// TIA Portal V20 export
FUNCTION_BLOCK "AdjRight"   // FB530, FBD
{ S7_Optimized_Access := 'TRUE' }
// stored: AutoNumber false, MemoryReserve 100, SetENOAutomatically false
   VAR
      Var { ExternalAccessible := 'False'; ExternalVisible := 'False'; ExternalWritable := 'False'} : "TypeVar";
      Cmd { ExternalAccessible := 'False'; ExternalVisible := 'False'; ExternalWritable := 'False'} : "TypeCmd";
      Enc { ExternalAccessible := 'False'; ExternalVisible := 'False'; ExternalWritable := 'False'} : "SysCounterFast";
      Pos { ExternalAccessible := 'False'; ExternalVisible := 'False'; ExternalWritable := 'False'} : "SysPos";
      AdjSlow { ExternalAccessible := 'False'; ExternalVisible := 'False'; ExternalWritable := 'False'} : "SysMotor";
      AdjFast { ExternalAccessible := 'False'; ExternalVisible := 'False'; ExternalWritable := 'False'} : "SysLinMotC1150";
      TAutoOn { ExternalAccessible := 'False'; ExternalVisible := 'False'; ExternalWritable := 'False'} : TON_TIME;
      TAutoTarPosManOn { ExternalAccessible := 'False'; ExternalVisible := 'False'; ExternalWritable := 'False'} : TON_TIME;
      T { ExternalAccessible := 'False'; ExternalVisible := 'False'; ExternalWritable := 'False'} : Array[1..5] of IEC_TIMER;
      adjFastPnSlaveOff { ExternalAccessible := 'False'; ExternalVisible := 'False'; ExternalWritable := 'False'} : "SysPnSlaveDeactivate";
      tarOld { ExternalAccessible := 'False'; ExternalVisible := 'False'; ExternalWritable := 'False'} : DInt;
      autoTarPosMan { ExternalAccessible := 'False'; ExternalVisible := 'False'; ExternalWritable := 'False'} : Bool;
      setValueEnc { ExternalAccessible := 'False'; ExternalVisible := 'False'; ExternalWritable := 'False'} : Bool;
      autoRef { ExternalAccessible := 'False'; ExternalVisible := 'False'; ExternalWritable := 'False'} : Bool;
      posOld { ExternalAccessible := 'False'; ExternalVisible := 'False'; ExternalWritable := 'False'} : Real;
      posDiff { ExternalAccessible := 'False'; ExternalVisible := 'False'; ExternalWritable := 'False'} : Real;
   END_VAR
   VAR_TEMP
      CtrlPc : Struct
         ackErr : Bool;
         manModeActive : Bool;
         manP : Bool;
         manM : Bool;
         manRefRun : Bool;
      END_STRUCT;
      CtrlLinMot : Struct
         mode : Int;
         target : Real;
         speed : Real;
         acc : Real;
         dec : Real;
         jerk : Real;
         autoRef : Bool;
      END_STRUCT;
      refPosDiff : DInt;
      offsetNoStd : Real;
      refPosDiffCalib : DInt;
      modeCalib : Int;
      disMechanicToZero : Int;   // distance mechanic part right to zero [mm]
   END_VAR
   VAR_TEMP   // added for the SCL form of the ladder/FBD networks
      _w1 : Bool;
   END_VAR
BEGIN

REGION Network 1 (SCL): offset for no standard calibration
   (* 
   normally the distance from camera to board should be 550mm
   for special application the distance is different
   the distance can be changed in the goldeneye program
   if its different then 550mm a offset will be added
   *)
   #offsetNoStd := 0.0;
   IF "ComRd".Data.Right.RefPosToBoard <> 550 THEN
       #offsetNoStd := (DINT_TO_REAL("ComRd".Data.Right.RefPosToBoard) - 550.0);
   ELSE
       #offsetNoStd := 0.0;
   END_IF;
END_REGION

REGION Network 2 (SCL): calibration value for offset
   (* 
   modus for calibartion
   camera must be referenced first
   mode 1 -->   the camera must be moved manually to position 550mm from board and
                 then press "Set Nullpoint"
   mode 2 -->   the camera must be moved to a other position and
                 then must be measured from the calibration tool to the camera and
                 this value must be putted in after pressing "Set Nullpoint"
   *)         
   #disMechanicToZero := 870; 
   #modeCalib := 2;
   IF #modeCalib = 1 THEN
       #refPosDiffCalib := "ComRd".Data.Right.TargetPos;
   ELSIF #modeCalib = 2 THEN
       #refPosDiffCalib := (#disMechanicToZero * 10) - ("ComRd".Data.Right.CalibratePos + 5500);
   END_IF;
END_REGION

REGION Network 3 (SCL): calibration value from pc
   "ComSd".Data.Right.SetCalibratePosOk := FALSE;

   IF "ComRd".Data.Right.SetCalibratePos THEN

       IF "G".Cfg.adjRightActive THEN
           #refPosDiff := REAL_TO_DINT("Enc"."8BC1.R".act * 10.0) - #refPosDiffCalib;
       ELSIF "G".Cfg.adjRightActiveLinMot THEN
           #refPosDiff := REAL_TO_DINT("Enc"."8U1.R".act * 10.0) - #refPosDiffCalib;
       END_IF;

       "Ref".adjRightCalOffset := #refPosDiff;
       "ComSd".Data.Right.SetCalibratePosOk := TRUE;

   END_IF;
END_REGION

REGION Network 4 (SCL): target position
   #Cmd.target := "G".Batch.width / 2.0;
   IF "G".Cfg.modeBoardPassing = 1 AND ("G".Cfg.modeDimension = 2 OR "G".Cfg.modeDimension = 4) AND NOT "G".Batch.stdActive THEN
       #Cmd.target := "G".Batch.width / 2.0 + ("G".Batch.widthMeasure - "G".Batch.width);
   END_IF;

   IF "G".Cfg.modeBoardPassing = 3 AND ("G".Cfg.modeDimension = 2 OR "G".Cfg.modeDimension = 4) AND NOT "G".Batch.stdActive THEN
       #Cmd.target :=  "G".Batch.senRightVal;
   END_IF;

   IF #autoTarPosMan THEN
       #Cmd.target := DINT_TO_REAL("ComRd".Data.Right.TargetPos) / 10.0;
   END_IF;

   "Ref".adjRightTar := #Cmd.target + (DINT_TO_REAL("Ref".adjRightCalOffset) / 10.0) + #offsetNoStd - "Enc"."8B1.B".offset;
END_REGION

REGION Network 5 (SCL): data from pc
   IF NOT "G".errComPc THEN
       #CtrlPc.manModeActive := "ComRd".Data.Right.ManModeActive;
       #CtrlPc.manP := "ComRd".Data.Right.ManPlus;
       #CtrlPc.manM := "ComRd".Data.Right.ManMinus;
       #CtrlPc.manRefRun := "ComRd".Data.Right.ManRefRun;
   ELSE
       #CtrlPc.manModeActive := TRUE;
       #CtrlPc.manP := FALSE;
       #CtrlPc.manM := FALSE;
       #CtrlPc.manRefRun := FALSE;
   END_IF;
   #CtrlPc.ackErr := "G".ack;
END_REGION

REGION Network 6: off
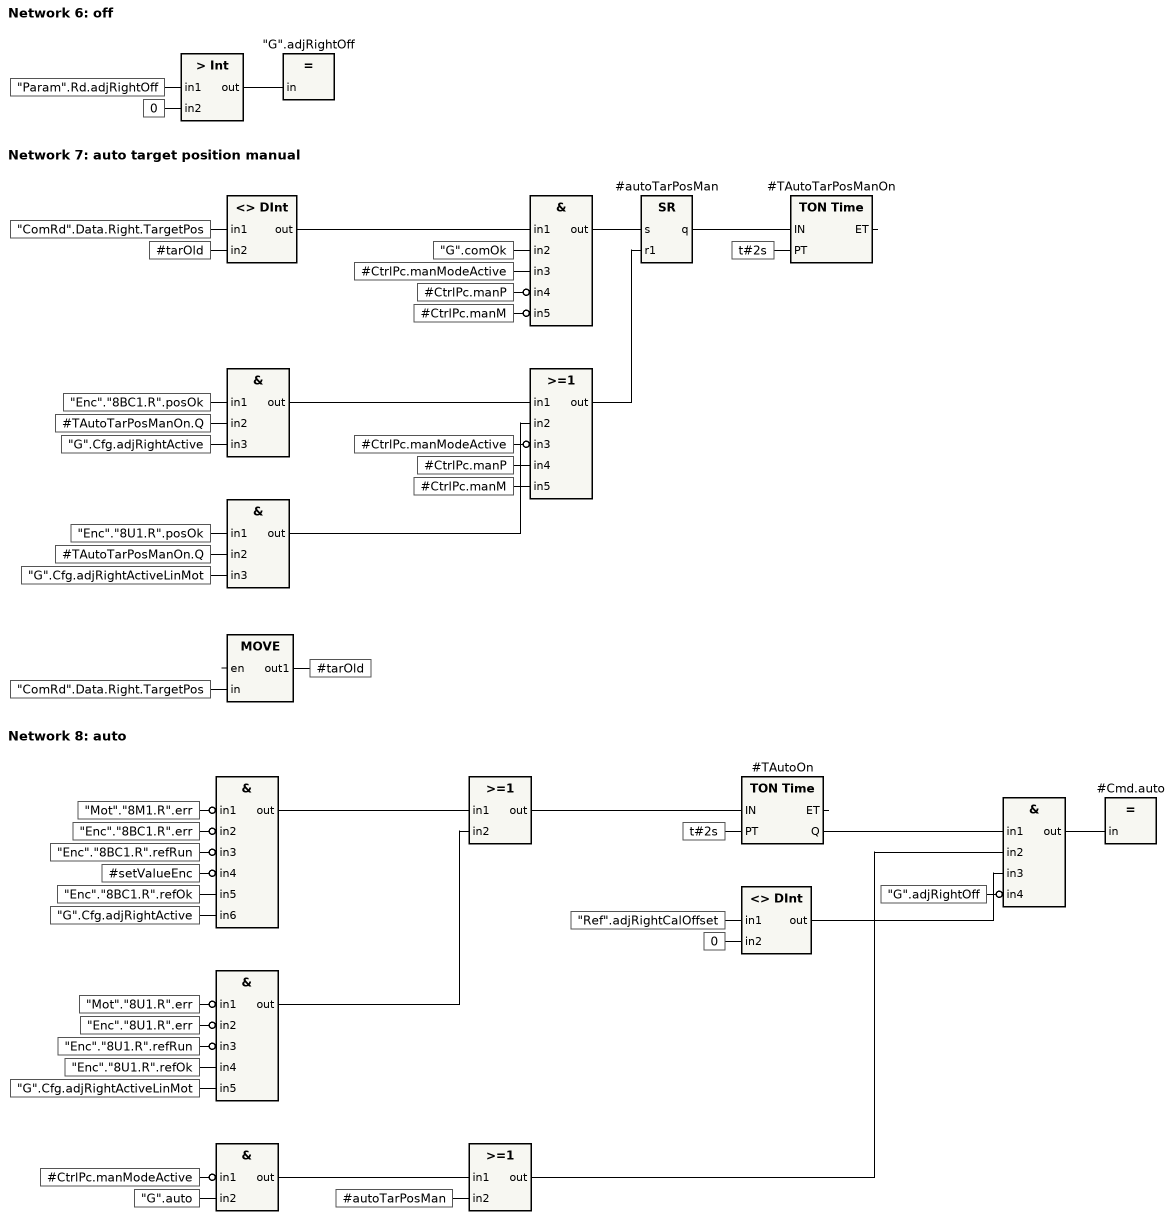
   "G".adjRightOff := "Param".Rd.adjRightOff > 0;
END_REGION

REGION Network 7: auto target position manual
   IF ("ComRd".Data.Right.TargetPos <> #tarOld) AND "G".comOk AND #CtrlPc.manModeActive AND NOT #CtrlPc.manP AND NOT #CtrlPc.manM THEN
       #autoTarPosMan := TRUE;   // SR flip-flop
   END_IF;
   IF ("Enc"."8BC1.R".posOk AND #TAutoTarPosManOn.Q AND "G".Cfg.adjRightActive) OR ("Enc"."8U1.R".posOk AND #TAutoTarPosManOn.Q AND "G".Cfg.adjRightActiveLinMot) OR NOT #CtrlPc.manModeActive OR #CtrlPc.manP OR #CtrlPc.manM THEN
       #autoTarPosMan := FALSE;
   END_IF;
   #TAutoTarPosManOn(IN := #autoTarPosMan, PT := t#2s);   // TON
   #tarOld := "ComRd".Data.Right.TargetPos;
END_REGION

REGION Network 8: auto
   #TAutoOn(IN := (NOT "Mot"."8M1.R".err AND NOT "Enc"."8BC1.R".err AND NOT "Enc"."8BC1.R".refRun AND NOT #setValueEnc AND "Enc"."8BC1.R".refOk AND "G".Cfg.adjRightActive) OR (NOT "Mot"."8U1.R".err AND NOT "Enc"."8U1.R".err AND NOT "Enc"."8U1.R".refRun AND "Enc"."8U1.R".refOk AND "G".Cfg.adjRightActiveLinMot),   // TON
            PT := t#2s);
   #Cmd.auto := #TAutoOn.Q AND ((NOT #CtrlPc.manModeActive AND "G".auto) OR #autoTarPosMan) AND ("Ref".adjRightCalOffset <> 0) AND NOT "G".adjRightOff;
END_REGION

REGION Network 9: manual
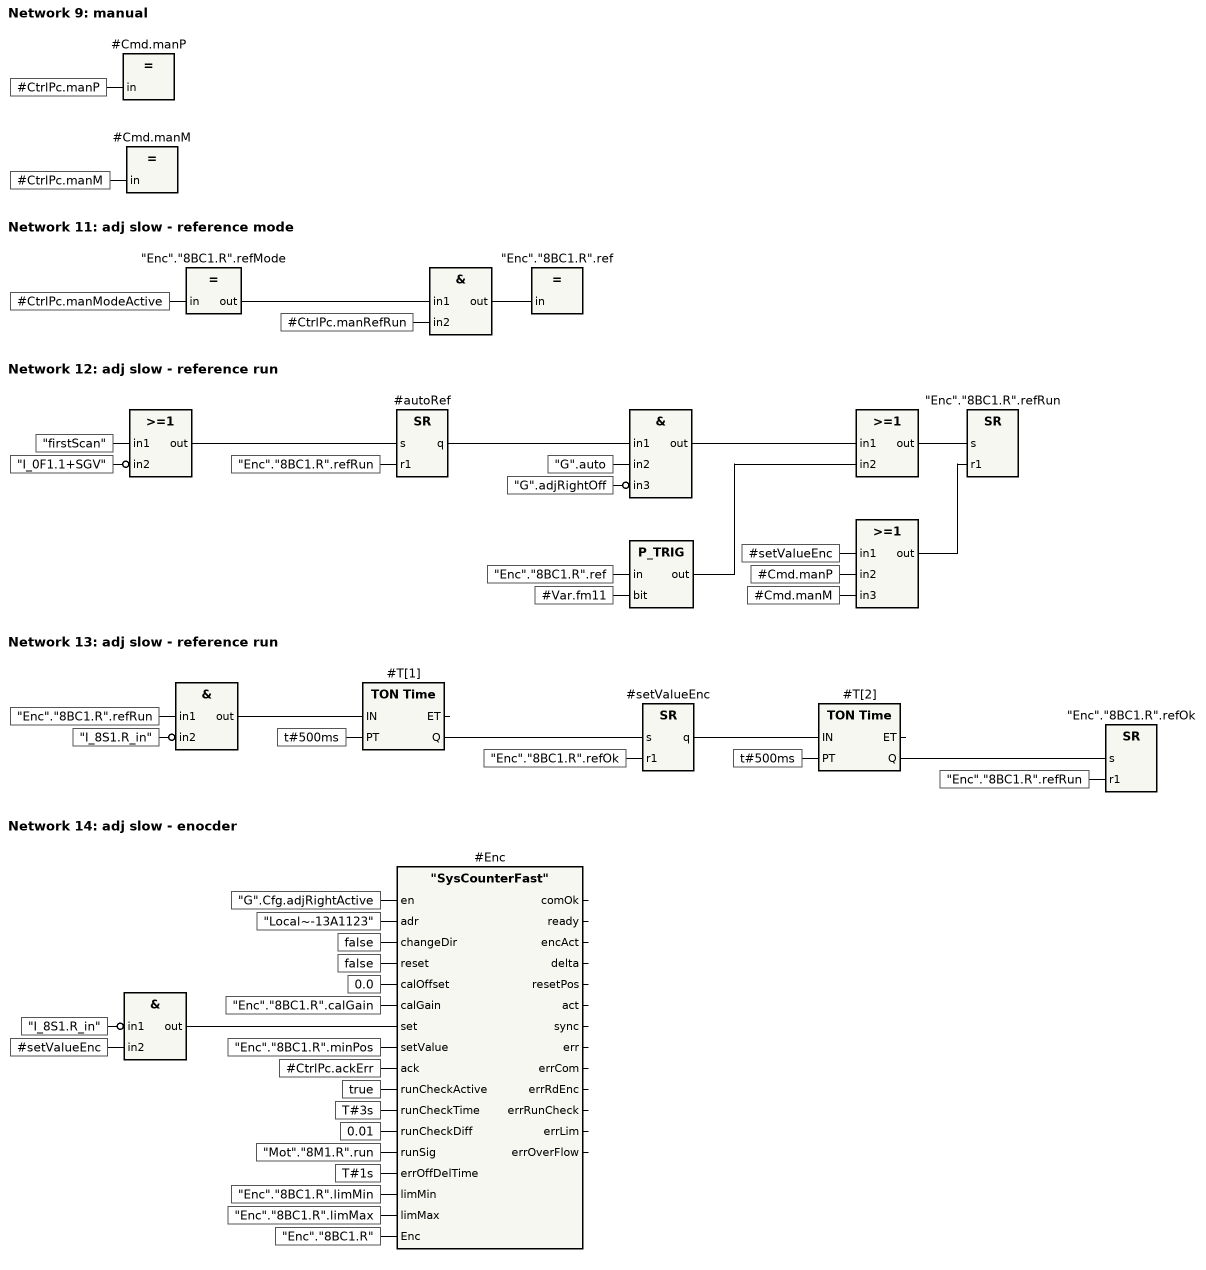
   #Cmd.manP := #CtrlPc.manP;
   #Cmd.manM := #CtrlPc.manM;
END_REGION

REGION Network 10 (SCL): adj slow - calibration value
   "Enc"."8BC1.R".calGain := -0.0275;

   "Enc"."8BC1.R".minPos := 10.0;
   "Enc"."8BC1.R".maxPos := 210.0;

   "Enc"."8BC1.R".limMin := "Enc"."8BC1.R".minPos - 5.0;
   "Enc"."8BC1.R".limMax := "Enc"."8BC1.R".maxPos + 5.0;

   "Enc"."8BC1.R".tarMinPos := "Enc"."8BC1.R".minPos + 0.0;
   "Enc"."8BC1.R".tarMaxPos := "Enc"."8BC1.R".maxPos - 0.0;
END_REGION

REGION Network 11: adj slow - reference mode
   "Enc"."8BC1.R".refMode := #CtrlPc.manModeActive;
   "Enc"."8BC1.R".ref := #CtrlPc.manModeActive AND #CtrlPc.manRefRun;
END_REGION

REGION Network 12: adj slow - reference run
   IF "firstScan" OR NOT "I_0F1.1+SGV" THEN
       #autoRef := TRUE;   // SR flip-flop
   END_IF;
   IF "Enc"."8BC1.R".refRun THEN #autoRef := FALSE; END_IF;
   #_w1 := "Enc"."8BC1.R".ref AND NOT #Var.fm11;   // rising edge
   #Var.fm11 := "Enc"."8BC1.R".ref;
   IF (#autoRef AND "G".auto AND NOT "G".adjRightOff) OR #_w1 THEN
       "Enc"."8BC1.R".refRun := TRUE;   // SR flip-flop
   END_IF;
   IF #setValueEnc OR #Cmd.manP OR #Cmd.manM THEN "Enc"."8BC1.R".refRun := FALSE; END_IF;
END_REGION

REGION Network 13: adj slow - reference run
   #T[1].TON(IN := "Enc"."8BC1.R".refRun AND NOT "I_8S1.R_in", PT := t#500ms);
   IF #T[1].Q THEN
       #setValueEnc := TRUE;   // SR flip-flop
   END_IF;
   IF "Enc"."8BC1.R".refOk THEN #setValueEnc := FALSE; END_IF;
   #T[2].TON(IN := #setValueEnc, PT := t#500ms);
   IF #T[2].Q THEN
       "Enc"."8BC1.R".refOk := TRUE;   // SR flip-flop
   END_IF;
   IF "Enc"."8BC1.R".refRun THEN "Enc"."8BC1.R".refOk := FALSE; END_IF;
END_REGION

REGION Network 14: adj slow - enocder
   IF "G".Cfg.adjRightActive THEN
       #Enc(adr := "Local~-13A1123",   // "SysCounterFast"
            changeDir := false,
            reset := false,
            calOffset := 0.0,
            calGain := "Enc"."8BC1.R".calGain,
            set := NOT "I_8S1.R_in" AND #setValueEnc,
            setValue := "Enc"."8BC1.R".minPos,
            ack := #CtrlPc.ackErr,
            runCheckActive := true,
            runCheckTime := T#3s,
            runCheckDiff := 0.01,
            runSig := "Mot"."8M1.R".run,
            errOffDelTime := T#1s,
            limMin := "Enc"."8BC1.R".limMin,
            limMax := "Enc"."8BC1.R".limMax,
            Enc := "Enc"."8BC1.R");
   END_IF;
END_REGION

REGION Network 15: adj slow - pos
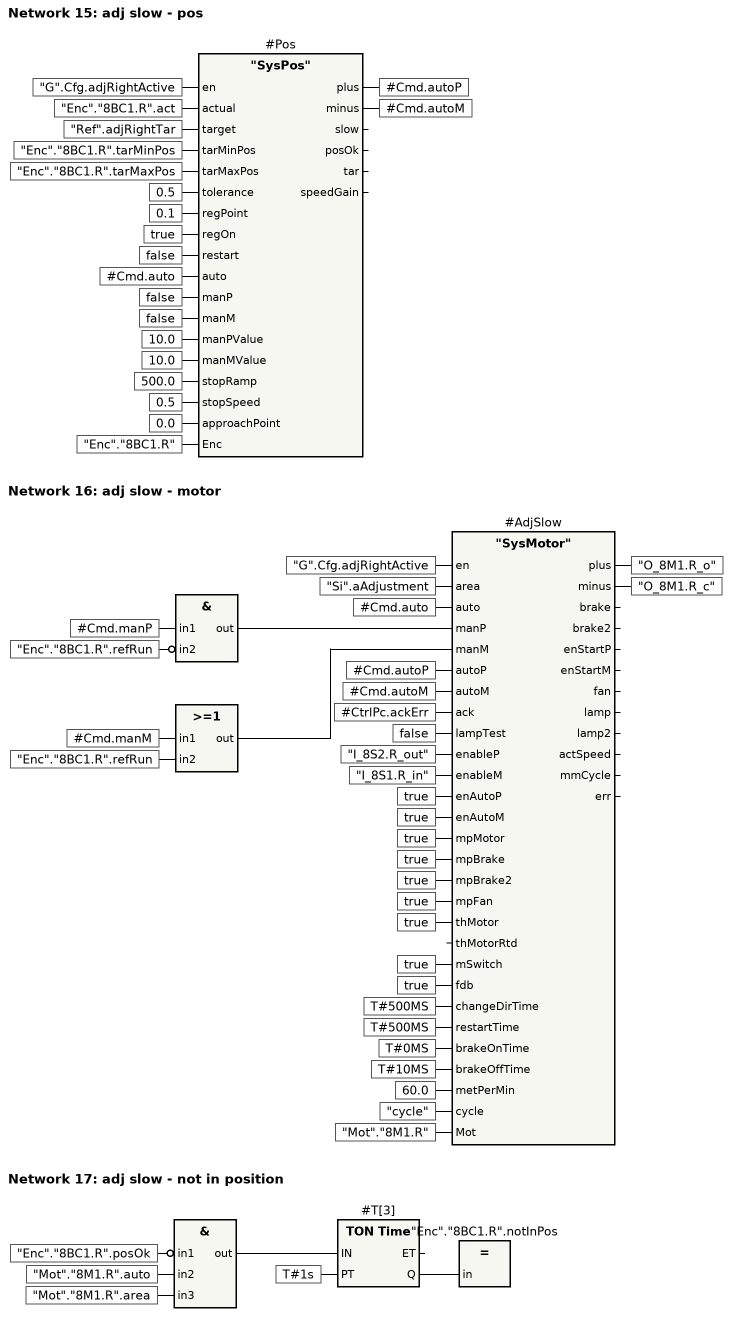
   IF "G".Cfg.adjRightActive THEN
       #Pos(actual := "Enc"."8BC1.R".act,   // "SysPos"
            target := "Ref".adjRightTar,
            tarMinPos := "Enc"."8BC1.R".tarMinPos,
            tarMaxPos := "Enc"."8BC1.R".tarMaxPos,
            tolerance := 0.5,
            regPoint := 0.1,
            regOn := true,
            restart := false,
            auto := #Cmd.auto,
            manP := false,
            manM := false,
            manPValue := 10.0,
            manMValue := 10.0,
            stopRamp := 500.0,
            stopSpeed := 0.5,
            approachPoint := 0.0,
            Enc := "Enc"."8BC1.R",
            plus => #Cmd.autoP,
            minus => #Cmd.autoM);
   END_IF;
END_REGION

REGION Network 16: adj slow - motor
   IF "G".Cfg.adjRightActive THEN
       #AdjSlow(area := "Si".aAdjustment,   // "SysMotor"
                auto := #Cmd.auto,
                manP := #Cmd.manP AND NOT "Enc"."8BC1.R".refRun,
                manM := #Cmd.manM OR "Enc"."8BC1.R".refRun,
                autoP := #Cmd.autoP,
                autoM := #Cmd.autoM,
                ack := #CtrlPc.ackErr,
                lampTest := false,
                enableP := "I_8S2.R_out",
                enableM := "I_8S1.R_in",
                enAutoP := true,
                enAutoM := true,
                mpMotor := true,
                mpBrake := true,
                mpBrake2 := true,
                mpFan := true,
                thMotor := true,
                mSwitch := true,
                fdb := true,
                changeDirTime := T#500MS,
                restartTime := T#500MS,
                brakeOnTime := T#0MS,
                brakeOffTime := T#10MS,
                metPerMin := 60.0,
                cycle := "cycle",
                Mot := "Mot"."8M1.R",
                plus => "O_8M1.R_o",
                minus => "O_8M1.R_c");
   END_IF;
END_REGION

REGION Network 17: adj slow - not in position
   #T[3].TON(IN := NOT "Enc"."8BC1.R".posOk AND "Mot"."8M1.R".auto AND "Mot"."8M1.R".area, PT := T#1s);
   "Enc"."8BC1.R".notInPos := #T[3].Q;
END_REGION

REGION Network 18: adj slow - sensor monitoring
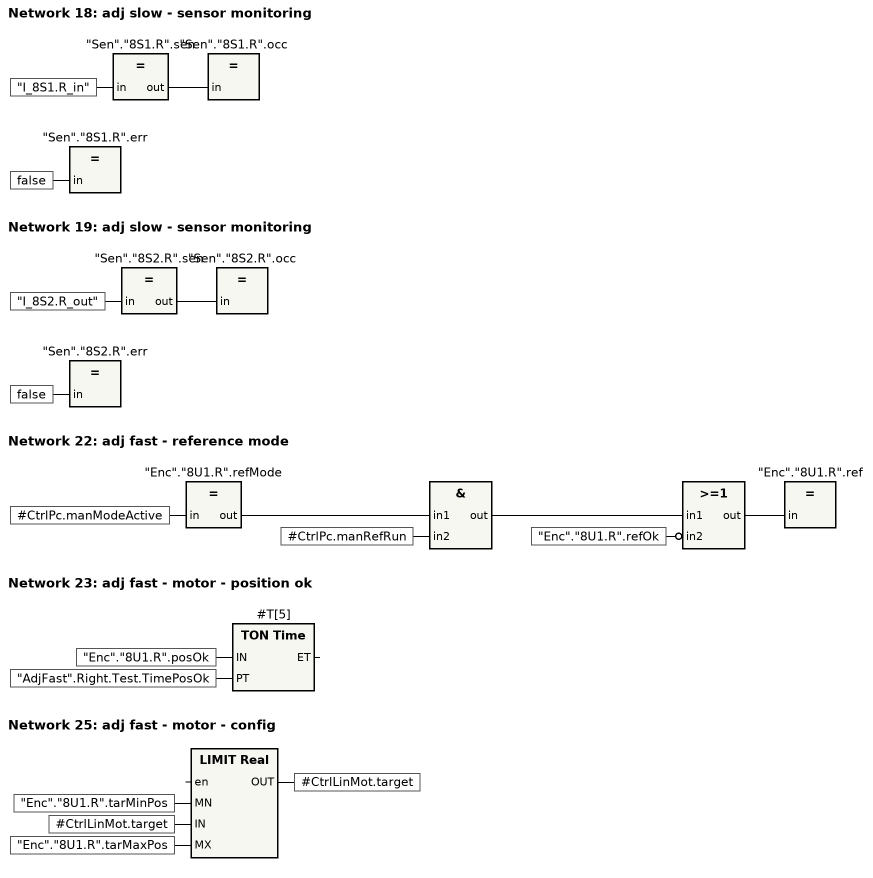
   "Sen"."8S1.R".sen := "I_8S1.R_in";
   "Sen"."8S1.R".occ := "I_8S1.R_in";
   "Sen"."8S1.R".err := false;
END_REGION

REGION Network 19: adj slow - sensor monitoring
   "Sen"."8S2.R".sen := "I_8S2.R_out";
   "Sen"."8S2.R".occ := "I_8S2.R_out";
   "Sen"."8S2.R".err := false;
END_REGION

REGION Network 21 (SCL): adj fast - calibration value
   "Enc"."8U1.R".calGain := 1.0;

   "Enc"."8U1.R".minPos := 5.0;
   "Enc"."8U1.R".maxPos := 155.0;

   "Enc"."8U1.R".limMin := "Enc"."8U1.R".minPos - 5.0;
   "Enc"."8U1.R".limMax := "Enc"."8U1.R".maxPos + 5.0;

   "Enc"."8U1.R".tarMinPos := "Enc"."8U1.R".minPos + 0.0;
   "Enc"."8U1.R".tarMaxPos := "Enc"."8U1.R".maxPos - 0.0;
END_REGION

REGION Network 22: adj fast - reference mode
   "Enc"."8U1.R".refMode := #CtrlPc.manModeActive;
   "Enc"."8U1.R".ref := (#CtrlPc.manModeActive AND #CtrlPc.manRefRun) OR NOT "Enc"."8U1.R".refOk;
END_REGION

REGION Network 23: adj fast - motor - position ok
   #T[5].TON(IN := "Enc"."8U1.R".posOk, PT := "AdjFast".Right.Test.TimePosOk);
END_REGION

REGION Network 24 (SCL): adj fast - motor - config

   //############################################################
   // min            5     mm
   // max          155     mm

   // speed        02      m/s
   // acc/dec      24      m/s2
   // jerk         450     m/s3

   // mode         BestehornVAJ
   //############################################################

   // only testmode for plc
   IF "AdjFast".Right.Test.ModeActive AND NOT #CtrlPc.manModeActive THEN
       IF "AdjFast".Right.Test.TarPos = "AdjFast".Right.Test.TarPos1 AND #T[5].Q THEN
           "AdjFast".Right.Test.TarPos := "AdjFast".Right.Test.TarPos2;
       ELSIF "AdjFast".Right.Test.TarPos = "AdjFast".Right.Test.TarPos2 AND #T[5].Q THEN
           "AdjFast".Right.Test.TarPos := "AdjFast".Right.Test.TarPos1;
       END_IF;
       "Ref".adjRightTar := "AdjFast".Right.Test.TarPos;
   END_IF;

   // active mode
   #CtrlLinMot.mode := 3;
   #CtrlLinMot.target := "Ref".adjRightTar;
   #CtrlLinMot.speed := 2.0;
   #CtrlLinMot.acc := 24.0;
   #CtrlLinMot.dec := 0.0;
   #CtrlLinMot.jerk := 450.0;

   // only testmode for plc
   IF "AdjFast".Right.Mode = 1 THEN
       #CtrlLinMot.mode := 1;
       #CtrlLinMot.target := "AdjFast".Right.VAI.Par1;
       #CtrlLinMot.speed := "AdjFast".Right.VAI.Par2;
       #CtrlLinMot.acc := "AdjFast".Right.VAI.Par3;
       #CtrlLinMot.dec := "AdjFast".Right.VAI.Par4;
       #CtrlLinMot.jerk := 0.0;
   ELSIF "AdjFast".Right.Mode = 2 THEN
       #CtrlLinMot.mode := 2;
       #CtrlLinMot.target := "AdjFast".Right.SinVA.Par1;
       #CtrlLinMot.speed := "AdjFast".Right.SinVA.Par2;
       #CtrlLinMot.acc := "AdjFast".Right.SinVA.Par3;
       #CtrlLinMot.dec := 0.0;
       #CtrlLinMot.jerk := 0.0;
   ELSIF "AdjFast".Right.Mode = 3 THEN
       #CtrlLinMot.mode := 3;
       #CtrlLinMot.target := "AdjFast".Right.BestehornVAJ.Par1;
       #CtrlLinMot.speed := "AdjFast".Right.BestehornVAJ.Par2;
       #CtrlLinMot.acc := "AdjFast".Right.BestehornVAJ.Par3;
       #CtrlLinMot.dec := 0.0;
       #CtrlLinMot.jerk := "AdjFast".Right.BestehornVAJ.Par4;
   END_IF;
END_REGION

REGION Network 25: adj fast - motor - config
   #CtrlLinMot.target := LIMIT(MN := "Enc"."8U1.R".tarMinPos, IN := #CtrlLinMot.target, MX := "Enc"."8U1.R".tarMaxPos);
END_REGION

REGION Network 26: adj fast - motor
   // #CtrlLinMot.target
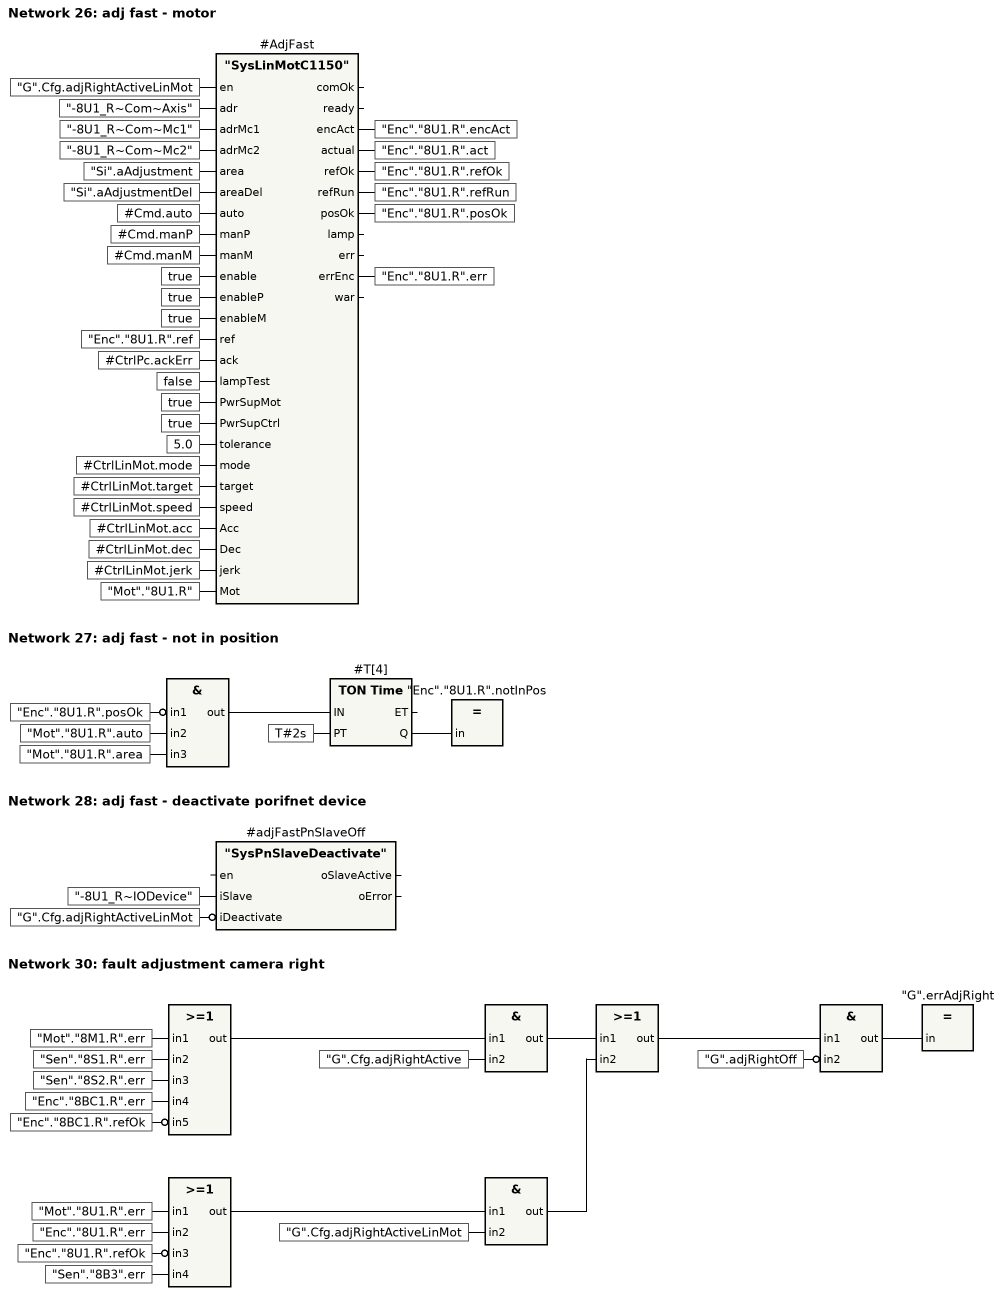
   IF "G".Cfg.adjRightActiveLinMot THEN
       #AdjFast(adr := "-8U1_R~Com~Axis",   // "SysLinMotC1150"
                adrMc1 := "-8U1_R~Com~Mc1",
                adrMc2 := "-8U1_R~Com~Mc2",
                area := "Si".aAdjustment,
                areaDel := "Si".aAdjustmentDel,
                auto := #Cmd.auto,
                manP := #Cmd.manP,
                manM := #Cmd.manM,
                enable := true,
                enableP := true,
                enableM := true,
                ref := "Enc"."8U1.R".ref,
                ack := #CtrlPc.ackErr,
                lampTest := false,
                PwrSupMot := true,
                PwrSupCtrl := true,
                tolerance := 5.0,
                mode := #CtrlLinMot.mode,
                target := #CtrlLinMot.target,
                speed := #CtrlLinMot.speed,
                Acc := #CtrlLinMot.acc,
                Dec := #CtrlLinMot.dec,
                jerk := #CtrlLinMot.jerk,
                Mot := "Mot"."8U1.R",
                encAct => "Enc"."8U1.R".encAct,
                actual => "Enc"."8U1.R".act,
                refOk => "Enc"."8U1.R".refOk,
                refRun => "Enc"."8U1.R".refRun,
                posOk => "Enc"."8U1.R".posOk,
                errEnc => "Enc"."8U1.R".err);
   END_IF;
END_REGION

REGION Network 27: adj fast - not in position
   #T[4].TON(IN := NOT "Enc"."8U1.R".posOk AND "Mot"."8U1.R".auto AND "Mot"."8U1.R".area, PT := T#2s);
   "Enc"."8U1.R".notInPos := #T[4].Q;
END_REGION

REGION Network 28: adj fast - deactivate porifnet device
   #adjFastPnSlaveOff(iSlave := "-8U1_R~IODevice", iDeactivate := NOT "G".Cfg.adjRightActiveLinMot);   // "SysPnSlaveDeactivate"
END_REGION

REGION Network 30: fault adjustment camera right
   "G".errAdjRight := ((("Mot"."8M1.R".err OR "Sen"."8S1.R".err OR "Sen"."8S2.R".err OR "Enc"."8BC1.R".err OR NOT "Enc"."8BC1.R".refOk) AND "G".Cfg.adjRightActive) OR (("Mot"."8U1.R".err OR "Enc"."8U1.R".err OR NOT "Enc"."8U1.R".refOk OR "Sen"."8B3".err) AND "G".Cfg.adjRightActiveLinMot)) AND NOT "G".adjRightOff;
END_REGION

REGION Network 31 (SCL): data to pc
   IF "G".Cfg.adjRightActive THEN
       "Ref".adjRightAct := REAL_TO_DINT("Enc"."8BC1.R".act * 10.0) - "Ref".adjRightCalOffset - REAL_TO_DINT(#offsetNoStd * 10.0);
       "ComSd".Data.Right.ActualEncPos := REAL_TO_DINT("Enc"."8BC1.R".act * 10.0);
       "ComSd".Data.Right.ActualPos :=  "Ref".adjRightAct;
       "ComSd".Data.Right.LimitSwitchMin := "Sen"."8S1.R".sen;
       "ComSd".Data.Right.LimitSwitchMax := "Sen"."8S2.R".sen;
       "ComSd".Data.Right.Err := "Mot"."8M1.R".err;
       "ComSd".Data.Right.ErrEnc := "Enc"."8BC1.R".err;
       "ComSd".Data.Right.PosOk := "Enc"."8BC1.R".posOk;
       "ComSd".Data.Right.Plus := "Mot"."8M1.R".plus;
       "ComSd".Data.Right.Minus := "Mot"."8M1.R".minus;
       "ComSd".Data.Right.refRun := "Enc"."8BC1.R".refRun;
       "ComSd".Data.Right.refOk := "Enc"."8BC1.R".refOk;
   ELSIF  "G".Cfg.adjRightActiveLinMot THEN
       "Ref".adjRightAct := REAL_TO_DINT("Enc"."8U1.R".act * 10.0) - "Ref".adjRightCalOffset - REAL_TO_DINT(#offsetNoStd * 10.0);
       "ComSd".Data.Right.ActualEncPos := REAL_TO_DINT("Enc"."8U1.R".act * 10.0);
       "ComSd".Data.Right.ActualPos :=  "Ref".adjRightAct;
       "ComSd".Data.Right.LimitSwitchMin := TRUE;
       "ComSd".Data.Right.LimitSwitchMax := TRUE;
       "ComSd".Data.Right.Err := "Mot"."8U1.R".err;
       "ComSd".Data.Right.ErrEnc := "Enc"."8U1.R".err;
       "ComSd".Data.Right.PosOk := "Enc"."8U1.R".posOk;
       "ComSd".Data.Right.Plus := "Mot"."8U1.R".plus;
       "ComSd".Data.Right.Minus := "Mot"."8U1.R".minus;
       "ComSd".Data.Right.refRun := "Enc"."8U1.R".refRun;
       "ComSd".Data.Right.refOk := "Enc"."8U1.R".refOk;
   ELSE
       "ComSd".Data.Right.ActualEncPos := 0;
       "ComSd".Data.Right.ActualPos := 0;
       "ComSd".Data.Right.LimitSwitchMin := FALSE;
       "ComSd".Data.Right.LimitSwitchMax := FALSE;
       "ComSd".Data.Right.Err := FALSE;
       "ComSd".Data.Right.ErrEnc := FALSE;
       "ComSd".Data.Right.PosOk := TRUE;
       "ComSd".Data.Right.Plus := FALSE;
       "ComSd".Data.Right.Minus := FALSE;
       "ComSd".Data.Right.refRun := FALSE;
       "ComSd".Data.Right.refOk := TRUE;
   END_IF;
END_REGION

REGION Network 32: current monitoring - auto
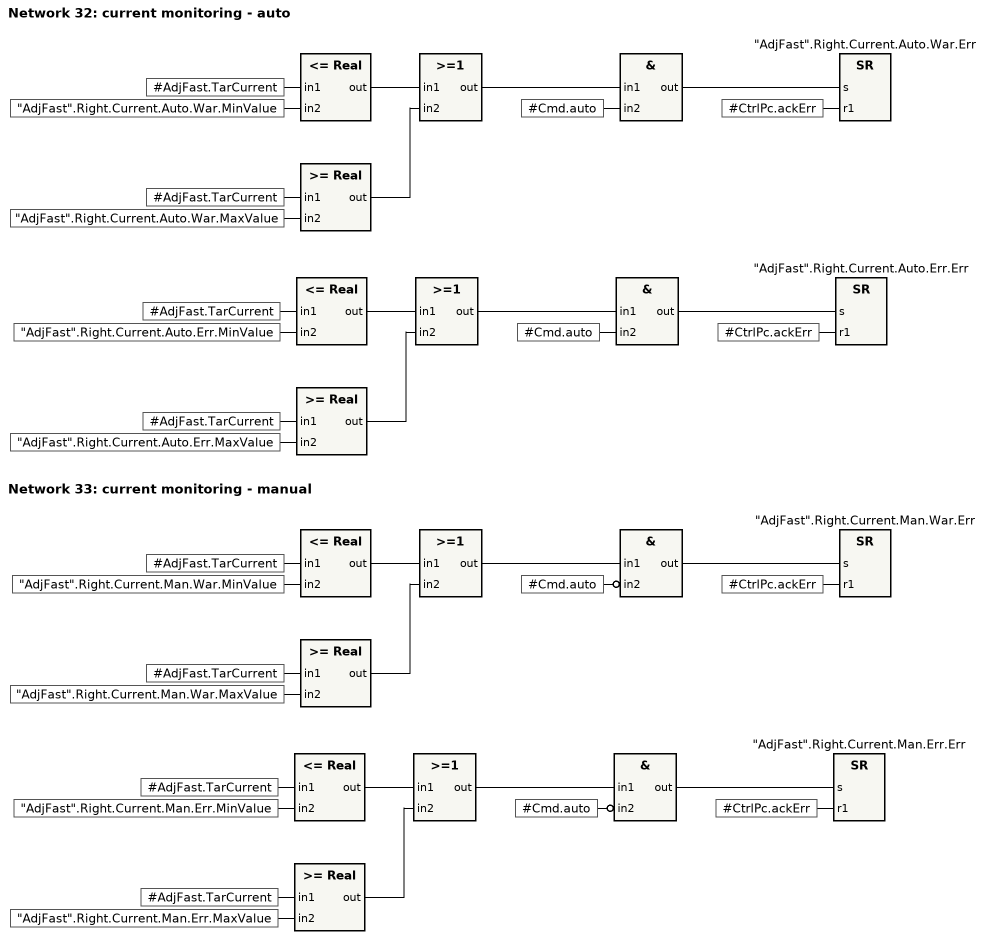
   IF ((#AdjFast.TarCurrent <= "AdjFast".Right.Current.Auto.War.MinValue) OR (#AdjFast.TarCurrent >= "AdjFast".Right.Current.Auto.War.MaxValue)) AND #Cmd.auto THEN
       "AdjFast".Right.Current.Auto.War.Err := TRUE;   // SR flip-flop
   END_IF;
   IF #CtrlPc.ackErr THEN "AdjFast".Right.Current.Auto.War.Err := FALSE; END_IF;
   IF ((#AdjFast.TarCurrent <= "AdjFast".Right.Current.Auto.Err.MinValue) OR (#AdjFast.TarCurrent >= "AdjFast".Right.Current.Auto.Err.MaxValue)) AND #Cmd.auto THEN
       "AdjFast".Right.Current.Auto.Err.Err := TRUE;   // SR flip-flop
   END_IF;
   IF #CtrlPc.ackErr THEN "AdjFast".Right.Current.Auto.Err.Err := FALSE; END_IF;
END_REGION

REGION Network 33: current monitoring - manual
   IF ((#AdjFast.TarCurrent <= "AdjFast".Right.Current.Man.War.MinValue) OR (#AdjFast.TarCurrent >= "AdjFast".Right.Current.Man.War.MaxValue)) AND NOT #Cmd.auto THEN
       "AdjFast".Right.Current.Man.War.Err := TRUE;   // SR flip-flop
   END_IF;
   IF #CtrlPc.ackErr THEN "AdjFast".Right.Current.Man.War.Err := FALSE; END_IF;
   IF ((#AdjFast.TarCurrent <= "AdjFast".Right.Current.Man.Err.MinValue) OR (#AdjFast.TarCurrent >= "AdjFast".Right.Current.Man.Err.MaxValue)) AND NOT #Cmd.auto THEN
       "AdjFast".Right.Current.Man.Err.Err := TRUE;   // SR flip-flop
   END_IF;
   IF #CtrlPc.ackErr THEN "AdjFast".Right.Current.Man.Err.Err := FALSE; END_IF;
END_REGION
END_FUNCTION_BLOCK
